// TIA Portal project "automated warehouse" (V15)
// Vorlageprojekt für das Buch mit Zielsystem S7-1200

(* hardware
DEVICE "S7-1200-Station_1"  S7-1200 Station
   slot 0: "Baugruppenträger_0"  Rack  V1.0
   slot 1: "PLC_1"  CPU 1211C DC/DC/DC  6ES7 211-1AE40-0XB0  V4.1
*)

// ===== PLC "PLC_1"  CPU 1211C DC/DC/DC =====

VAR_GLOBAL   // PLC tag table "Standard-Variablentabelle"
   "at entry" AT %I0.0 : Bool;
   "at load" AT %I0.1 : Bool;
   "at left" AT %I0.2 : Bool;
   "at middle" AT %I0.3 : Bool;
   "at right" AT %I0.4 : Bool;
   "at unload" AT %I0.5 : Bool;
   "at exit" AT %I0.6 : Bool;
   "moving x" AT %I0.7 : Bool;
   "moving z" AT %I1.0 : Bool;
   "start" AT %I1.1 : Bool;
   "reset" AT %I1.2 : Bool;
   "stop" AT %I1.3 : Bool;
   "emergency stop" AT %I1.4 : Bool;
   "auto" AT %I1.5 : Bool;
   "entry conveyor" AT %Q0.0 : Bool;
   "load conveyor" AT %Q0.1 : Bool;
   "forks left" AT %Q0.2 : Bool;
   "forks right" AT %Q0.3 : Bool;
   "lift" AT %Q0.4 : Bool;
   "unload conveyor" AT %Q0.5 : Bool;
   "exit conveyor" AT %Q0.6 : Bool;
   "start light" AT %Q0.7 : Bool;
   "reset light" AT %Q1.0 : Bool;
   "stop light" AT %Q1.1 : Bool;
   "palet sayısı" AT %MW100 : Int;
   "Tag_1" AT %QD100 : DWord;
   "Tag_2" AT %QD30 : DWord;
   "Tag_3" AT %M99.0 : Bool;
   "Tag_4" AT %QW30 : Int;
   "Tag_5" AT %QD1 : DWord;
   "Tag_6" AT %M10.2 : Bool;
   "Tag_7" AT %M10.3 : Bool;
   "Tag_8" AT %M6.0 : Bool;
   "Tag_9" AT %QW75 : Word;
   "Tag_10" AT %QD75 : DWord;
   "son" AT %M80.0 : Bool;
END_VAR

// folder: System blocks/Program resources

DATA_BLOCK "asansör kalkıs geciktirme"   // DB1
{ S7_Optimized_Access := 'TRUE' }
AUTHOR : Simatic
FAMILY : IEC
NAME : IEC_TMR
VERSION : 1.0
// stored: InstanceOfName IEC_TIMER
"IEC_TIMER"
BEGIN
END_DATA_BLOCK

DATA_BLOCK "IEC_Timer_0_DB"   // DB2
{ S7_Optimized_Access := 'TRUE' }
AUTHOR : Simatic
FAMILY : IEC
NAME : IEC_TMR
VERSION : 1.0
// stored: InstanceOfName IEC_TIMER
"IEC_TIMER"
BEGIN
END_DATA_BLOCK

DATA_BLOCK "palet sayıcı"   // DB3
{ S7_Optimized_Access := 'TRUE' }
AUTHOR : Simatic
FAMILY : IEC
NAME : CNTR
VERSION : 1.0
// stored: InstanceOfName IEC_COUNTER
"IEC_COUNTER"
BEGIN
END_DATA_BLOCK

DATA_BLOCK "IEC_Counter_0_DB"   // DB4
{ S7_Optimized_Access := 'TRUE' }
AUTHOR : Simatic
FAMILY : IEC
NAME : CNTR
VERSION : 1.0
// stored: InstanceOfName IEC_COUNTER
"IEC_COUNTER"
BEGIN
END_DATA_BLOCK

DATA_BLOCK "sağ taraf bekleme"   // DB5
{ S7_Optimized_Access := 'TRUE' }
AUTHOR : Simatic
FAMILY : IEC
NAME : IEC_TMR
VERSION : 1.0
// stored: InstanceOfName IEC_TIMER
"IEC_TIMER"
BEGIN
END_DATA_BLOCK

DATA_BLOCK "gecikme"   // DB6
{ S7_Optimized_Access := 'TRUE' }
AUTHOR : Simatic
FAMILY : IEC
NAME : IEC_TMR
VERSION : 1.0
// stored: InstanceOfName IEC_TIMER
"IEC_TIMER"
BEGIN
END_DATA_BLOCK

DATA_BLOCK "x bekleme"   // DB7
{ S7_Optimized_Access := 'TRUE' }
AUTHOR : Simatic
FAMILY : IEC
NAME : IEC_TMR
VERSION : 1.0
// stored: InstanceOfName IEC_TIMER
"IEC_TIMER"
BEGIN
END_DATA_BLOCK

DATA_BLOCK "indirme geciktirme"   // DB8
{ S7_Optimized_Access := 'TRUE' }
AUTHOR : Simatic
FAMILY : IEC
NAME : IEC_TMR
VERSION : 1.0
// stored: InstanceOfName IEC_TIMER
"IEC_TIMER"
BEGIN
END_DATA_BLOCK

DATA_BLOCK "indirme bekleme"   // DB9
{ S7_Optimized_Access := 'TRUE' }
AUTHOR : Simatic
FAMILY : IEC
NAME : IEC_TMR
VERSION : 1.0
// stored: InstanceOfName IEC_TIMER
"IEC_TIMER"
BEGIN
END_DATA_BLOCK

// folder: (top level)

FUNCTION "MHJ-PLC-Lab-Function-S71200" : Void   // FC9000, SCL
{ S7_Optimized_Access := 'TRUE' }
VERSION : 0.1
   VAR_TEMP
      rdTimeReturn : Int;
      outputTime : DTL;
      SyncVal : Byte;
      forVal : Int;
      forVal_2 : Int;
      Value : Byte;
   END_VAR
   VAR CONSTANT
      CompVal : Byte := 16#34;
      Value_01 : Byte := 16#11;
      Value_01_DW : DWord := 16#A165_D992;
      Value_02_DW : DWord := 16#58BE_4401;
   END_VAR
BEGIN

   #Value:=PEEK(area := 16#82,
        dbNumber := 0,
        byteOffset := 511);
   #Value := #Value + 1;

   POKE(area := 16#82,
        dbNumber := 0,
        byteOffset := 511,
        value := #Value);

   POKE(area:=16#81,
        dbNumber:=0,
        byteOffset:=1016,
        value:=#Value_01_DW);
   POKE(area := 16#81,
        dbNumber := 0,
        byteOffset := 1020,
        value := #Value_02_DW);

   POKE(area := 16#81,
        dbNumber := 0,
        byteOffset := 511,
        value := B#16#00);

   FOR #forVal := 0 TO 120 DO
       FOR #forVal_2:=0 TO 10 DO
           #rdTimeReturn:=RD_SYS_T(#outputTime);
           #rdTimeReturn := WR_SYS_T(#outputTime);
           #rdTimeReturn := RD_SYS_T(#outputTime);
           #rdTimeReturn := WR_SYS_T(#outputTime);
       END_FOR;
       #SyncVal:= PEEK(area := 16#81,
                      dbNumber := 0,
                      byteOffset := 511);
       IF #SyncVal = #CompVal THEN
          GOTO M_1;
       END_IF;
   END_FOR;
   RETURN;

   M_1:
   POKE(area := 16#81,
        dbNumber := 0,
        byteOffset := 511,
        value := B#16#0);
END_FUNCTION

ORGANIZATION_BLOCK "Main"   // OB1, LAD, ProgramCycle
TITLE = "Main Program Sweep (Cycle)"
{ S7_Optimized_Access := 'TRUE' }
VERSION : 0.1
   VAR_INPUT
      Initial_Call : Bool;   // Initial call of this OB
      Remanence : Bool;   // =True, if remanent data are available
   END_VAR
BEGIN

REGION Network 1
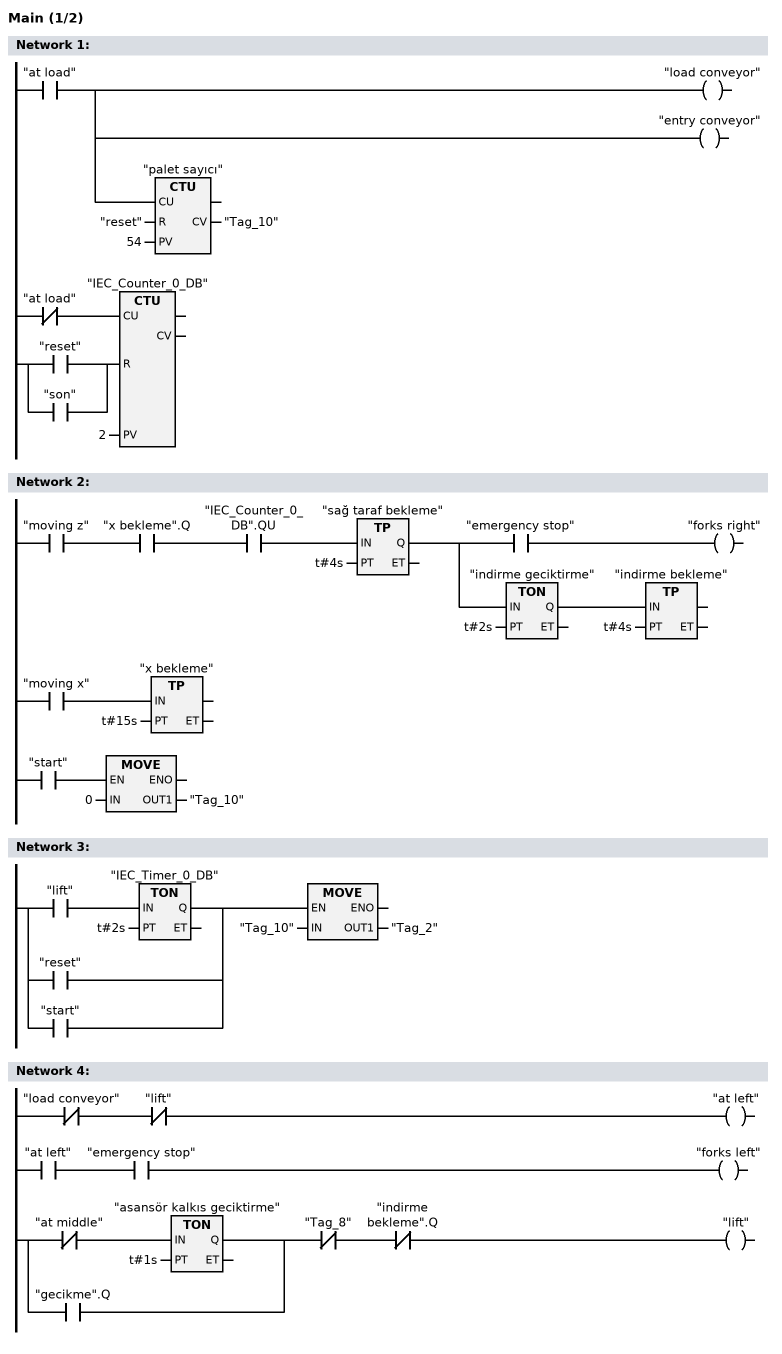
   "load conveyor" := "at load";
   "entry conveyor" := "at load";
   "palet sayıcı".CTU(CU := "at load", R := "reset", PV := 54, CV => "Tag_10");
   "IEC_Counter_0_DB".CTU(CU := NOT "at load", R := "reset" OR "son", PV := 2);
END_REGION

REGION Network 2
   "sağ taraf bekleme".TP(IN := "moving z" AND "x bekleme".Q AND "IEC_Counter_0_DB".QU, PT := t#4s);
   "forks right" := "sağ taraf bekleme".Q AND "emergency stop";
   "indirme geciktirme".TON(IN := "sağ taraf bekleme".Q, PT := t#2s);
   "indirme bekleme".TP(IN := "indirme geciktirme".Q, PT := t#4s);
   "x bekleme".TP(IN := "moving x", PT := t#15s);
   IF "start" THEN "Tag_10" := 0; END_IF;
END_REGION

REGION Network 3
   "IEC_Timer_0_DB".TON(IN := "lift", PT := t#2s);
   IF "IEC_Timer_0_DB".Q OR "reset" OR "start" THEN "Tag_2" := "Tag_10"; END_IF;
END_REGION

REGION Network 4
   "at left" := NOT "load conveyor" AND NOT "lift";
   "forks left" := "at left" AND "emergency stop";
   "asansör kalkıs geciktirme".TON(IN := NOT "at middle", PT := t#1s);
   "lift" := ("asansör kalkıs geciktirme".Q OR "gecikme".Q) AND NOT "Tag_8" AND NOT "indirme bekleme".Q;
END_REGION

REGION Network 5
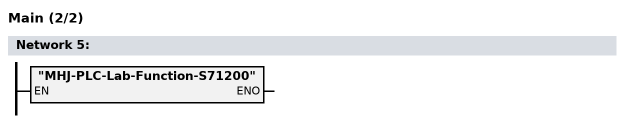
   RUNG wire#powerrail
      "MHJ-PLC-Lab-Function-S71200"()
   END_RUNG
   // the same network as SCL:
   "MHJ-PLC-Lab-Function-S71200"();
END_REGION
END_ORGANIZATION_BLOCK